// TIA Portal V20 export
DATA_BLOCK "LBP_MFuncDecListSignals"   // DB76
TITLE = M decoding acc. to list / Décodage M selon liste
{ S7_Optimized_Access := 'FALSE' }
AUTHOR : SINUMERIK
FAMILY : SINUMERIK_ONE
VERSION : 6.24
// Interface between user program and NCK, contains the signal list for the request and acknowledgment of the M functions configured with LBP_MFuncDecListConfig [DB75] / Interface entre programme utilisateur et NCK contient la liste des signaux pour la demande et l'acquittement des fonctions M configurées avec LBP_MFuncDecListConfig [DB75]
// stored: AutoNumber false
   VAR
      MSigGrp1 : Struct
         MSig : Array[0..15] of Bool;
      END_STRUCT;
      MSigGrp2 : Struct
         MSig : Array[0..15] of Bool;
      END_STRUCT;
      MSigGrp3 : Struct
         MSig : Array[0..15] of Bool;
      END_STRUCT;
      MSigGrp4 : Struct
         MSig : Array[0..15] of Bool;
      END_STRUCT;
      MSigGrp5 : Struct
         MSig : Array[0..15] of Bool;
      END_STRUCT;
      MSigGrp6 : Struct
         MSig : Array[0..15] of Bool;
      END_STRUCT;
      MSigGrp7 : Struct
         MSig : Array[0..15] of Bool;
      END_STRUCT;
      MSigGrp8 : Struct
         MSig : Array[0..15] of Bool;
      END_STRUCT;
      MSigGrp9 : Struct
         MSig : Array[0..15] of Bool;
      END_STRUCT;
      MSigGrp10 : Struct
         MSig : Array[0..15] of Bool;
      END_STRUCT;
      MSigGrp11 : Struct
         MSig : Array[0..15] of Bool;
      END_STRUCT;
      MSigGrp12 : Struct
         MSig : Array[0..15] of Bool;
      END_STRUCT;
      MSigGrp13 : Struct
         MSig : Array[0..15] of Bool;
      END_STRUCT;
      MSigGrp14 : Struct
         MSig : Array[0..15] of Bool;
      END_STRUCT;
      MSigGrp15 : Struct
         MSig : Array[0..15] of Bool;
      END_STRUCT;
      MSigGrp16 : Struct
         MSig : Array[0..15] of Bool;
      END_STRUCT;
   END_VAR
BEGIN
END_DATA_BLOCK
